TYPE ST_UserControlGrid_ToHmi :
STRUCT
	stButtonSave	: ST_HMI_BUTTON_OUT;
END_STRUCT
END_TYPE

(* stored: Version 1.1.0.1, ProductVersion 3.1.4024.11
   DUT ST_UserControlGrid_ToHmi: Id {e4cb23bf-7773-44c5-aecf-ae301cdcaa11} *)
